// TIA Portal V17 export
// export: Created 2024-09-02T12:50:23.3039212Z, ExportSetting WithDefaults, DisplayName Totally Integrated Automation Portal, DisplayVersion V17, DisplayName TIA Portal Openness, DisplayVersion V17, DisplayName TIA Portal Version Control Interface, DisplayVersion V17, DisplayName STEP 7 Professional, DisplayVersion V17, DisplayName STEP 7 Safety, DisplayVersion V17, DisplayName WinCC Professional, DisplayVersion V17
FUNCTION "AnwFC_Aveva_OP701" : Void   // FC35, LAD
{ S7_Optimized_Access := 'TRUE' }
VERSION : 0.1
// stored: AutoNumber true, IsIECCheckEnabled false, SetENOAutomatically false, UDAEnableTagReadback false
   VAR_TEMP
      Data_Ready : Bool;
      Pallet_Nr_Moved : Bool;
      Converted_Data : Real;
      tEKSLevelOK : Bool;
   END_VAR
   VAR CONSTANT
      cButtonNotActive : USInt := 0;
      cButtonActive : USInt := 1;
      cColorRed : USInt := 2;
      cColorGreen : USInt := 3;
      cMesOptionEmpty : USInt := 0;
      cMesReasonEmpty : String := '';
   END_VAR
   VAR_TEMP   // added for the SCL form of the ladder/FBD networks
      _w1 : Bool;
      _w2 : Bool;
      _w3 : Bool;
      _w4 : Bool;
   END_VAR
BEGIN

REGION Network 1: ################STEP 1 - Pallet arrive to station #################
END_REGION

REGION Network 2: Copy Nr of Pallet
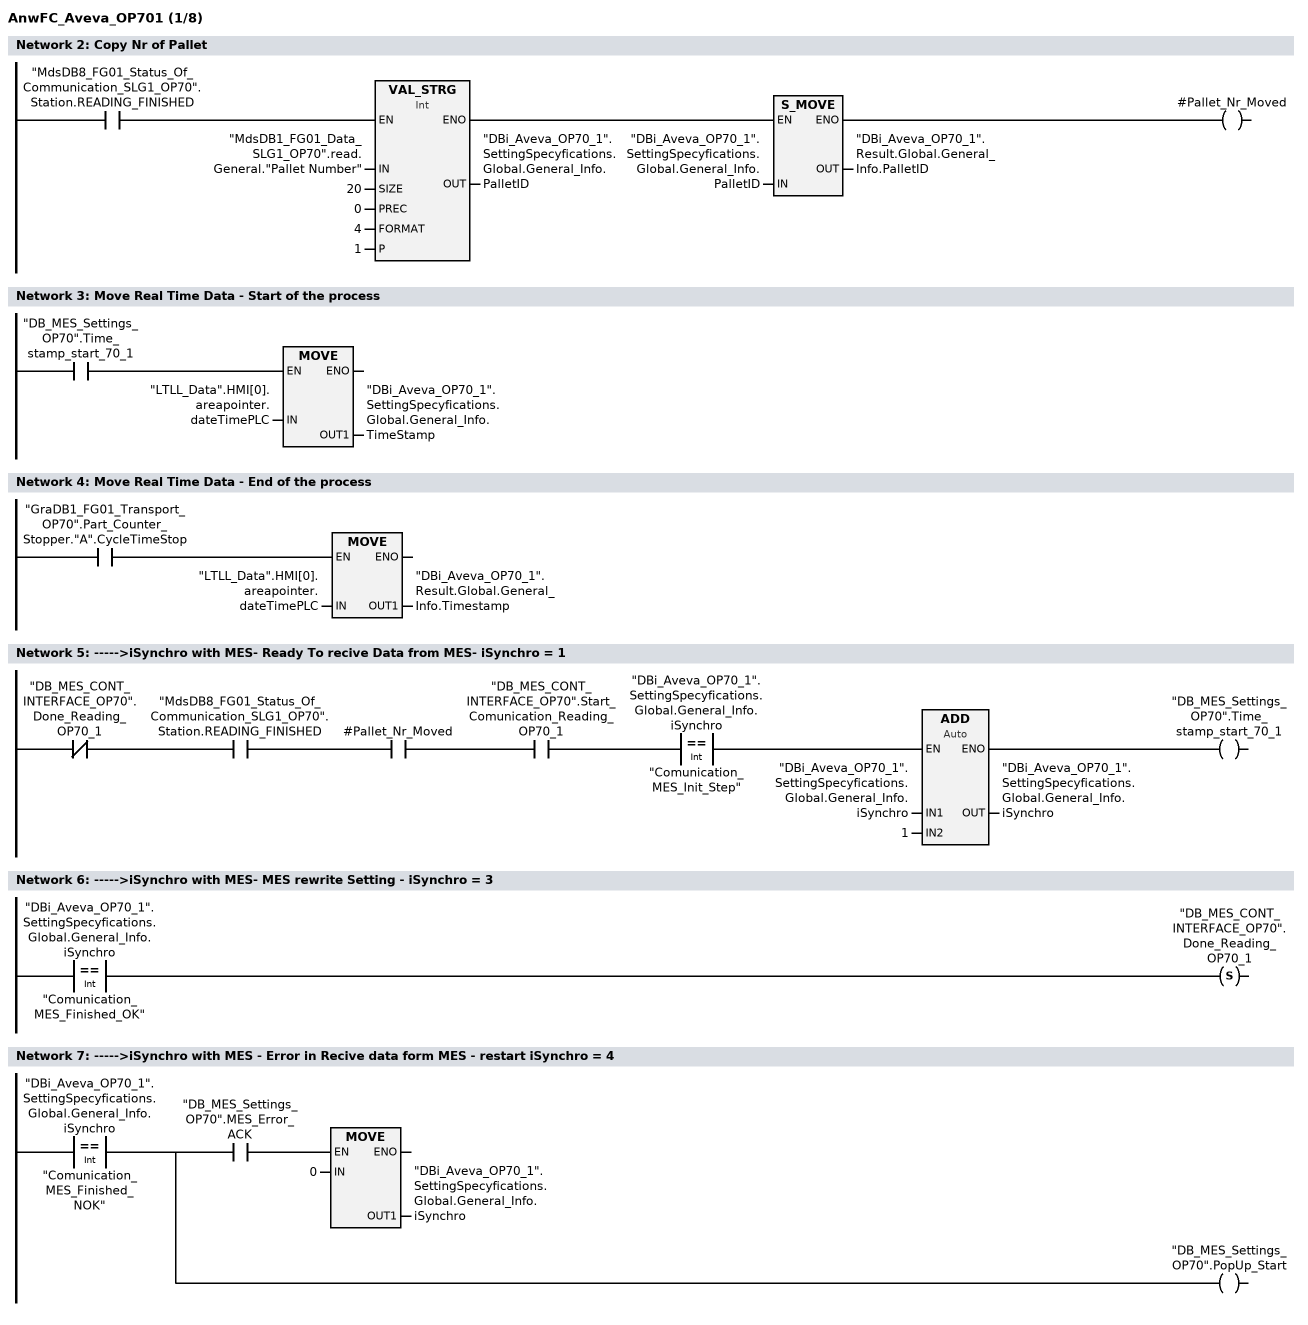
   RUNG wire#powerrail
      Contact( "MdsDB8_FG01_Status_Of_Communication_SLG1_OP70".Station.READING_FINISHED )
      { S7_Templates := "[value_type := Int, str_type := String]" } VAL_STRG(IN := "MdsDB1_FG01_Data_SLG1_OP70".read.General."Pallet Number", SIZE := 20, PREC := 0, FORMAT := 4, P := 1, OUT => "DBi_Aveva_OP70_1".SettingSpecyfications.Global.General_Info.PalletID)
      S_Move(in := "DBi_Aveva_OP70_1".SettingSpecyfications.Global.General_Info.PalletID, out => "DBi_Aveva_OP70_1".Result.Global.General_Info.PalletID)
      Coil( #Pallet_Nr_Moved )
   END_RUNG
   // the same network as SCL:
   VAL_STRG(EN := "MdsDB8_FG01_Status_Of_Communication_SLG1_OP70".Station.READING_FINISHED,
            IN := "MdsDB1_FG01_Data_SLG1_OP70".read.General."Pallet Number",
            SIZE := 20,
            PREC := 0,
            FORMAT := 4,
            P := 1,
            OUT => "DBi_Aveva_OP70_1".SettingSpecyfications.Global.General_Info.PalletID,
            ENO => #_w1);
   IF #_w1 THEN
       "DBi_Aveva_OP70_1".Result.Global.General_Info.PalletID := "DBi_Aveva_OP70_1".SettingSpecyfications.Global.General_Info.PalletID;
   END_IF;
   #Pallet_Nr_Moved := #_w1;
END_REGION

REGION Network 3: Move Real Time Data - Start of the process
   RUNG wire#powerrail
      Contact( "DB_MES_Settings_OP70".Time_stamp_start_70_1 )
      Move(in := "LTLL_Data".HMI[0].areapointer.dateTimePLC, out1 => "DBi_Aveva_OP70_1".SettingSpecyfications.Global.General_Info.TimeStamp)
   END_RUNG
   // the same network as SCL:
   IF "DB_MES_Settings_OP70".Time_stamp_start_70_1 THEN
       "DBi_Aveva_OP70_1".SettingSpecyfications.Global.General_Info.TimeStamp := "LTLL_Data".HMI[0].areapointer.dateTimePLC;
   END_IF;
END_REGION

REGION Network 4: Move Real Time Data - End of the process
   RUNG wire#powerrail
      Contact( "GraDB1_FG01_Transport_OP70".Part_Counter_Stopper."A".CycleTimeStop )
      Move(in := "LTLL_Data".HMI[0].areapointer.dateTimePLC, out1 => "DBi_Aveva_OP70_1".Result.Global.General_Info.Timestamp)
   END_RUNG
   // the same network as SCL:
   IF "GraDB1_FG01_Transport_OP70".Part_Counter_Stopper."A".CycleTimeStop THEN
       "DBi_Aveva_OP70_1".Result.Global.General_Info.Timestamp := "LTLL_Data".HMI[0].areapointer.dateTimePLC;
   END_IF;
END_REGION

REGION Network 5: ----->iSynchro with MES- Ready To recive Data from MES- iSynchro = 1
   RUNG wire#powerrail
      I_Contact( "DB_MES_CONT_INTERFACE_OP70".Done_Reading_OP70_1 )
      Contact( "MdsDB8_FG01_Status_Of_Communication_SLG1_OP70".Station.READING_FINISHED )
      Contact( #Pallet_Nr_Moved )
      Contact( "DB_MES_CONT_INTERFACE_OP70".Start_Comunication_Reading_OP70_1 )
      { S7_Templates := "SrcType := Int" } EQ_Contact(in1 := "DBi_Aveva_OP70_1".SettingSpecyfications.Global.General_Info.iSynchro, in2 := "Comunication_MES_Init_Step")
      Add(in1 := "DBi_Aveva_OP70_1".SettingSpecyfications.Global.General_Info.iSynchro, in2 := 1, out => "DBi_Aveva_OP70_1".SettingSpecyfications.Global.General_Info.iSynchro)
      Coil( "DB_MES_Settings_OP70".Time_stamp_start_70_1 )
   END_RUNG
   // the same network as SCL:
   #_w1 := NOT "DB_MES_CONT_INTERFACE_OP70".Done_Reading_OP70_1 AND "MdsDB8_FG01_Status_Of_Communication_SLG1_OP70".Station.READING_FINISHED AND #Pallet_Nr_Moved AND "DB_MES_CONT_INTERFACE_OP70".Start_Comunication_Reading_OP70_1 AND ("DBi_Aveva_OP70_1".SettingSpecyfications.Global.General_Info.iSynchro = "Comunication_MES_Init_Step");
   IF #_w1 THEN
       "DBi_Aveva_OP70_1".SettingSpecyfications.Global.General_Info.iSynchro := "DBi_Aveva_OP70_1".SettingSpecyfications.Global.General_Info.iSynchro + 1;
   END_IF;
   "DB_MES_Settings_OP70".Time_stamp_start_70_1 := #_w1;
END_REGION

REGION Network 6: ----->iSynchro with MES- MES rewrite Setting - iSynchro = 3
   RUNG wire#powerrail
      { S7_Templates := "SrcType := Int" } EQ_Contact(in1 := "DBi_Aveva_OP70_1".SettingSpecyfications.Global.General_Info.iSynchro, in2 := "Comunication_MES_Finished_OK")
      S_Coil( "DB_MES_CONT_INTERFACE_OP70".Done_Reading_OP70_1 )
   END_RUNG
   // the same network as SCL:
   IF "DBi_Aveva_OP70_1".SettingSpecyfications.Global.General_Info.iSynchro = "Comunication_MES_Finished_OK" THEN
       "DB_MES_CONT_INTERFACE_OP70".Done_Reading_OP70_1 := TRUE;
   END_IF;
END_REGION

REGION Network 7: ----->iSynchro with MES - Error in Recive data form MES - restart iSynchro = 4
   RUNG wire#powerrail
      { S7_Templates := "SrcType := Int" } EQ_Contact(in1 := "DBi_Aveva_OP70_1".SettingSpecyfications.Global.General_Info.iSynchro, in2 := "Comunication_MES_Finished_NOK")
      wire#w1
      Contact( "DB_MES_Settings_OP70".MES_Error_ACK )
      Move(in := 0, out1 => "DBi_Aveva_OP70_1".SettingSpecyfications.Global.General_Info.iSynchro)
   END_RUNG
   RUNG wire#w1
      Coil( "DB_MES_Settings_OP70".PopUp_Start )
   END_RUNG
   // the same network as SCL:
   #_w1 := "DBi_Aveva_OP70_1".SettingSpecyfications.Global.General_Info.iSynchro = "Comunication_MES_Finished_NOK";
   IF #_w1 AND "DB_MES_Settings_OP70".MES_Error_ACK THEN
       "DBi_Aveva_OP70_1".SettingSpecyfications.Global.General_Info.iSynchro := 0;
   END_IF;
   "DB_MES_Settings_OP70".PopUp_Start := #_w1;
END_REGION

REGION Network 8: ----->iSynchro with MES - End of Analyse - restart iSynchro = 0
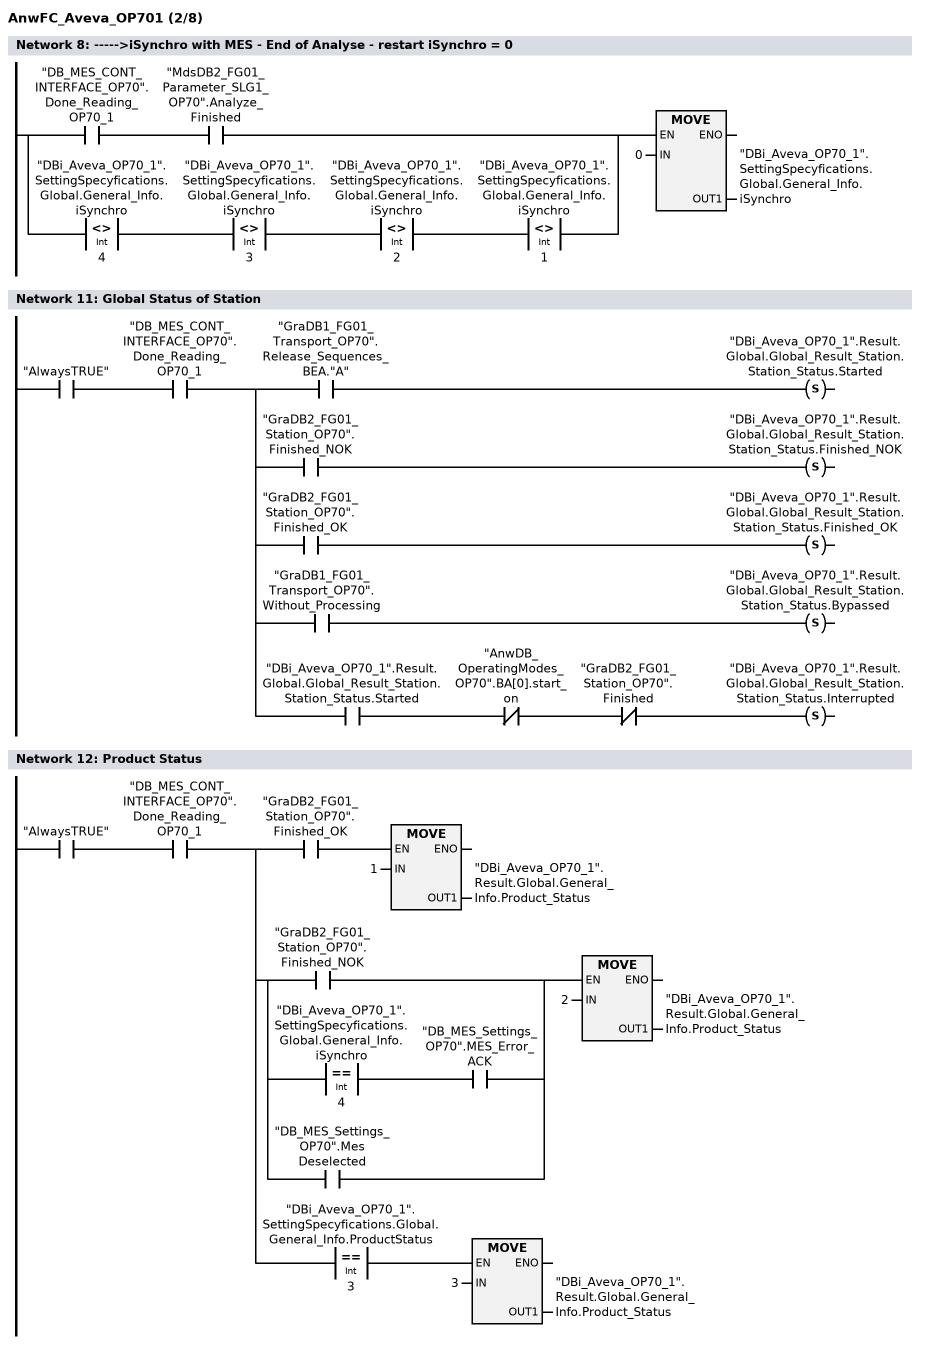
   RUNG wire#powerrail
      Contact( "DB_MES_CONT_INTERFACE_OP70".Done_Reading_OP70_1 )
      Contact( "MdsDB2_FG01_Parameter_SLG1_OP70".Analyze_Finished )
      wire#w1
      Move(in := 0, out1 => "DBi_Aveva_OP70_1".SettingSpecyfications.Global.General_Info.iSynchro)
   END_RUNG
   RUNG wire#powerrail
      { S7_Templates := "SrcType := Int" } NE_Contact(in1 := "DBi_Aveva_OP70_1".SettingSpecyfications.Global.General_Info.iSynchro, in2 := 4)
      { S7_Templates := "SrcType := Int" } NE_Contact(in1 := "DBi_Aveva_OP70_1".SettingSpecyfications.Global.General_Info.iSynchro, in2 := 3)
      { S7_Templates := "SrcType := Int" } NE_Contact(in1 := "DBi_Aveva_OP70_1".SettingSpecyfications.Global.General_Info.iSynchro, in2 := 2)
      { S7_Templates := "SrcType := Int" } NE_Contact(in1 := "DBi_Aveva_OP70_1".SettingSpecyfications.Global.General_Info.iSynchro, in2 := 1)
   END_RUNG wire#w1
   // the same network as SCL:
   IF ("DB_MES_CONT_INTERFACE_OP70".Done_Reading_OP70_1 AND "MdsDB2_FG01_Parameter_SLG1_OP70".Analyze_Finished) OR (("DBi_Aveva_OP70_1".SettingSpecyfications.Global.General_Info.iSynchro <> 4) AND ("DBi_Aveva_OP70_1".SettingSpecyfications.Global.General_Info.iSynchro <> 3) AND ("DBi_Aveva_OP70_1".SettingSpecyfications.Global.General_Info.iSynchro <> 2) AND ("DBi_Aveva_OP70_1".SettingSpecyfications.Global.General_Info.iSynchro <> 1)) THEN
       "DBi_Aveva_OP70_1".SettingSpecyfications.Global.General_Info.iSynchro := 0;
   END_IF;
END_REGION

REGION Network 9: ################STEP 2 - Move the Proce Data From Each Operation ################# / Status Proces 1
   // IN0 - Aktor ist abgewählt
   // IN1 - TAF ist angewählt
   // IN2 - Nacharbeit in Station
   // IN3 - Auftrag manuell vorgegeben
   // IN4 - Nacharbeit auf Standby-Platz
   // IN5 - Nacharbeit auf EAS-Platz
   // IN6 - TAF hat gearbeitet (Fertigmeldung)
   // IN7 - Bauteil wurde iO bearbeitet
END_REGION

REGION Network 10: ################STEP 2 - Move the Proce Data From Station ################# / Status Proces 1
   // IN0 - Aktor ist abgewählt
   // IN1 - TAF ist angewählt
   // IN2 - Nacharbeit in Station
   // IN3 - Auftrag manuell vorgegeben
   // IN4 - Nacharbeit auf Standby-Platz
   // IN5 - Nacharbeit auf EAS-Platz
   // IN6 - TAF hat gearbeitet (Fertigmeldung)
   // IN7 - Bauteil wurde iO bearbeitet
END_REGION

REGION Network 11: Global Status of Station
   RUNG wire#powerrail
      Contact( "AlwaysTRUE" )
      Contact( "DB_MES_CONT_INTERFACE_OP70".Done_Reading_OP70_1 )
      wire#w1
      Contact( "GraDB1_FG01_Transport_OP70".Release_Sequences_BEA."A" )
      S_Coil( "DBi_Aveva_OP70_1".Result.Global.Global_Result_Station.Station_Status.Started )
   END_RUNG
   RUNG wire#w1
      Contact( "GraDB2_FG01_Station_OP70".Finished_NOK )
      S_Coil( "DBi_Aveva_OP70_1".Result.Global.Global_Result_Station.Station_Status.Finished_NOK )
   END_RUNG
   RUNG wire#w1
      Contact( "GraDB2_FG01_Station_OP70".Finished_OK )
      S_Coil( "DBi_Aveva_OP70_1".Result.Global.Global_Result_Station.Station_Status.Finished_OK )
   END_RUNG
   RUNG wire#w1
      Contact( "GraDB1_FG01_Transport_OP70".Without_Processing )
      S_Coil( "DBi_Aveva_OP70_1".Result.Global.Global_Result_Station.Station_Status.Bypassed )
   END_RUNG
   RUNG wire#w1
      Contact( "DBi_Aveva_OP70_1".Result.Global.Global_Result_Station.Station_Status.Started )
      I_Contact( "AnwDB_OperatingModes_OP70".BA[0].start_on )
      I_Contact( "GraDB2_FG01_Station_OP70".Finished )
      S_Coil( "DBi_Aveva_OP70_1".Result.Global.Global_Result_Station.Station_Status.Interrupted )
   END_RUNG
   // the same network as SCL:
   #_w1 := "AlwaysTRUE" AND "DB_MES_CONT_INTERFACE_OP70".Done_Reading_OP70_1;
   IF #_w1 AND "GraDB1_FG01_Transport_OP70".Release_Sequences_BEA."A" THEN
       "DBi_Aveva_OP70_1".Result.Global.Global_Result_Station.Station_Status.Started := TRUE;
   END_IF;
   IF #_w1 AND "GraDB2_FG01_Station_OP70".Finished_NOK THEN
       "DBi_Aveva_OP70_1".Result.Global.Global_Result_Station.Station_Status.Finished_NOK := TRUE;
   END_IF;
   IF #_w1 AND "GraDB2_FG01_Station_OP70".Finished_OK THEN
       "DBi_Aveva_OP70_1".Result.Global.Global_Result_Station.Station_Status.Finished_OK := TRUE;
   END_IF;
   IF #_w1 AND "GraDB1_FG01_Transport_OP70".Without_Processing THEN
       "DBi_Aveva_OP70_1".Result.Global.Global_Result_Station.Station_Status.Bypassed := TRUE;
   END_IF;
   IF #_w1 AND "DBi_Aveva_OP70_1".Result.Global.Global_Result_Station.Station_Status.Started AND NOT "AnwDB_OperatingModes_OP70".BA[0].start_on AND NOT "GraDB2_FG01_Station_OP70".Finished THEN
       "DBi_Aveva_OP70_1".Result.Global.Global_Result_Station.Station_Status.Interrupted := TRUE;
   END_IF;
END_REGION

REGION Network 12: Product Status
   RUNG wire#powerrail
      Contact( "AlwaysTRUE" )
      Contact( "DB_MES_CONT_INTERFACE_OP70".Done_Reading_OP70_1 )
      wire#w1
      Contact( "GraDB2_FG01_Station_OP70".Finished_OK )
      Move(in := 1, out1 => "DBi_Aveva_OP70_1".Result.Global.General_Info.Product_Status)
   END_RUNG
   RUNG wire#w1
      Contact( "GraDB2_FG01_Station_OP70".Finished_NOK )
      wire#w2
      Move(in := 2, out1 => "DBi_Aveva_OP70_1".Result.Global.General_Info.Product_Status)
   END_RUNG
   RUNG wire#w1
      { S7_Templates := "SrcType := Int" } EQ_Contact(in1 := "DBi_Aveva_OP70_1".SettingSpecyfications.Global.General_Info.iSynchro, in2 := 4)
      Contact( "DB_MES_Settings_OP70".MES_Error_ACK )
   END_RUNG wire#w2
   RUNG wire#w1
      Contact( "DB_MES_Settings_OP70".MesDeselected )
   END_RUNG wire#w2
   RUNG wire#w1
      { S7_Templates := "SrcType := Int" } EQ_Contact(in1 := "DBi_Aveva_OP70_1".SettingSpecyfications.Global.General_Info.ProductStatus, in2 := 3)
      Move(in := 3, out1 => "DBi_Aveva_OP70_1".Result.Global.General_Info.Product_Status)
   END_RUNG
   // the same network as SCL:
   #_w1 := "AlwaysTRUE" AND "DB_MES_CONT_INTERFACE_OP70".Done_Reading_OP70_1;
   IF #_w1 AND "GraDB2_FG01_Station_OP70".Finished_OK THEN
       "DBi_Aveva_OP70_1".Result.Global.General_Info.Product_Status := 1;
   END_IF;
   IF #_w1 AND ("GraDB2_FG01_Station_OP70".Finished_NOK OR (("DBi_Aveva_OP70_1".SettingSpecyfications.Global.General_Info.iSynchro = 4) AND "DB_MES_Settings_OP70".MES_Error_ACK) OR "DB_MES_Settings_OP70".MesDeselected) THEN
       "DBi_Aveva_OP70_1".Result.Global.General_Info.Product_Status := 2;
   END_IF;
   IF #_w1 AND ("DBi_Aveva_OP70_1".SettingSpecyfications.Global.General_Info.ProductStatus = 3) THEN
       "DBi_Aveva_OP70_1".Result.Global.General_Info.Product_Status := 3;
   END_IF;
END_REGION

REGION Network 13: ################ STEP 3 - Prepare Isynchro for MES in result area #################
END_REGION

REGION Network 14: ----->iSynchro with MES- Ready To copy Data to MES- - iSynchro = 1
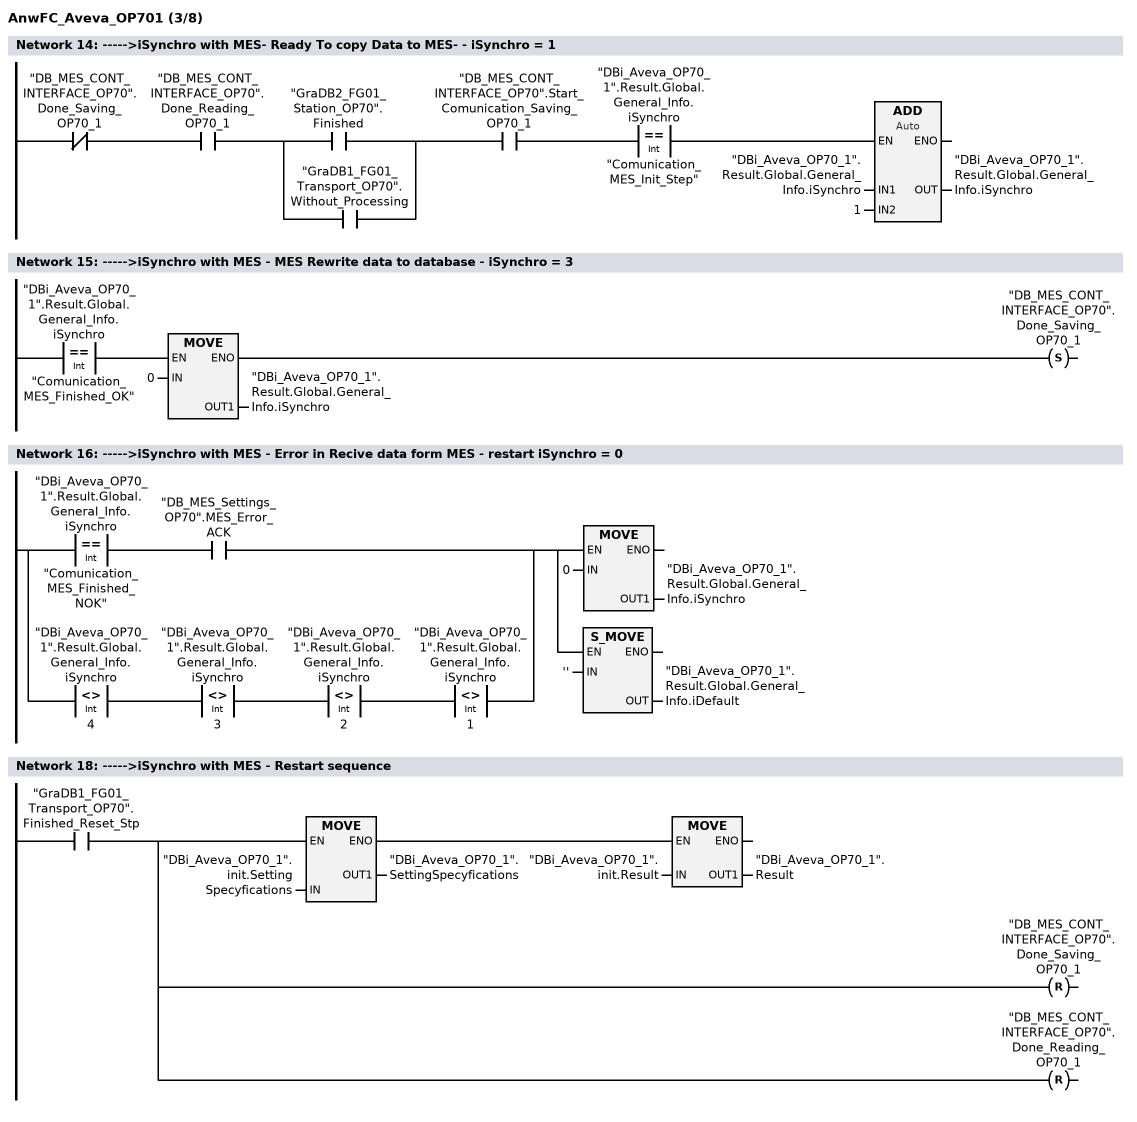
   RUNG wire#powerrail
      I_Contact( "DB_MES_CONT_INTERFACE_OP70".Done_Saving_OP70_1 )
      Contact( "DB_MES_CONT_INTERFACE_OP70".Done_Reading_OP70_1 )
      wire#w1
      Contact( "GraDB2_FG01_Station_OP70".Finished )
      wire#w2
      Contact( "DB_MES_CONT_INTERFACE_OP70".Start_Comunication_Saving_OP70_1 )
      { S7_Templates := "SrcType := Int" } EQ_Contact(in1 := "DBi_Aveva_OP70_1".Result.Global.General_Info.iSynchro, in2 := "Comunication_MES_Init_Step")
      Add(in1 := "DBi_Aveva_OP70_1".Result.Global.General_Info.iSynchro, in2 := 1, out => "DBi_Aveva_OP70_1".Result.Global.General_Info.iSynchro)
   END_RUNG
   RUNG wire#w1
      Contact( "GraDB1_FG01_Transport_OP70".Without_Processing )
   END_RUNG wire#w2
   // the same network as SCL:
   IF NOT "DB_MES_CONT_INTERFACE_OP70".Done_Saving_OP70_1 AND "DB_MES_CONT_INTERFACE_OP70".Done_Reading_OP70_1 AND ("GraDB2_FG01_Station_OP70".Finished OR "GraDB1_FG01_Transport_OP70".Without_Processing) AND "DB_MES_CONT_INTERFACE_OP70".Start_Comunication_Saving_OP70_1 AND ("DBi_Aveva_OP70_1".Result.Global.General_Info.iSynchro = "Comunication_MES_Init_Step") THEN
       "DBi_Aveva_OP70_1".Result.Global.General_Info.iSynchro := "DBi_Aveva_OP70_1".Result.Global.General_Info.iSynchro + 1;
   END_IF;
END_REGION

REGION Network 15: ----->iSynchro with MES - MES Rewrite data to database - iSynchro = 3
   RUNG wire#powerrail
      { S7_Templates := "SrcType := Int" } EQ_Contact(in1 := "DBi_Aveva_OP70_1".Result.Global.General_Info.iSynchro, in2 := "Comunication_MES_Finished_OK")
      Move(in := 0, out1 => "DBi_Aveva_OP70_1".Result.Global.General_Info.iSynchro)
      S_Coil( "DB_MES_CONT_INTERFACE_OP70".Done_Saving_OP70_1 )
   END_RUNG
   // the same network as SCL:
   #_w1 := "DBi_Aveva_OP70_1".Result.Global.General_Info.iSynchro = "Comunication_MES_Finished_OK";
   IF #_w1 THEN
       "DBi_Aveva_OP70_1".Result.Global.General_Info.iSynchro := 0;
       "DB_MES_CONT_INTERFACE_OP70".Done_Saving_OP70_1 := TRUE;
   END_IF;
END_REGION

REGION Network 16: ----->iSynchro with MES - Error in Recive data form MES - restart iSynchro = 0
   RUNG wire#powerrail
      { S7_Templates := "SrcType := Int" } EQ_Contact(in1 := "DBi_Aveva_OP70_1".Result.Global.General_Info.iSynchro, in2 := "Comunication_MES_Finished_NOK")
      Contact( "DB_MES_Settings_OP70".MES_Error_ACK )
      wire#w1
      Move(in := 0, out1 => "DBi_Aveva_OP70_1".Result.Global.General_Info.iSynchro)
   END_RUNG
   RUNG wire#powerrail
      { S7_Templates := "SrcType := Int" } NE_Contact(in1 := "DBi_Aveva_OP70_1".Result.Global.General_Info.iSynchro, in2 := 4)
      { S7_Templates := "SrcType := Int" } NE_Contact(in1 := "DBi_Aveva_OP70_1".Result.Global.General_Info.iSynchro, in2 := 3)
      { S7_Templates := "SrcType := Int" } NE_Contact(in1 := "DBi_Aveva_OP70_1".Result.Global.General_Info.iSynchro, in2 := 2)
      { S7_Templates := "SrcType := Int" } NE_Contact(in1 := "DBi_Aveva_OP70_1".Result.Global.General_Info.iSynchro, in2 := 1)
   END_RUNG wire#w1
   RUNG wire#w1
      S_Move(in := '', out => "DBi_Aveva_OP70_1".Result.Global.General_Info.iDefault)
   END_RUNG
   // the same network as SCL:
   #_w1 := (("DBi_Aveva_OP70_1".Result.Global.General_Info.iSynchro = "Comunication_MES_Finished_NOK") AND "DB_MES_Settings_OP70".MES_Error_ACK) OR (("DBi_Aveva_OP70_1".Result.Global.General_Info.iSynchro <> 4) AND ("DBi_Aveva_OP70_1".Result.Global.General_Info.iSynchro <> 3) AND ("DBi_Aveva_OP70_1".Result.Global.General_Info.iSynchro <> 2) AND ("DBi_Aveva_OP70_1".Result.Global.General_Info.iSynchro <> 1));
   IF #_w1 THEN
       "DBi_Aveva_OP70_1".Result.Global.General_Info.iSynchro := 0;
       "DBi_Aveva_OP70_1".Result.Global.General_Info.iDefault := '';
   END_IF;
END_REGION

REGION Network 17: ################ STEP3 - Restart all #################
END_REGION

REGION Network 18: ----->iSynchro with MES - Restart sequence
   RUNG wire#powerrail
      Contact( "GraDB1_FG01_Transport_OP70".Finished_Reset_Stp )
      wire#w1
      Move(in := "DBi_Aveva_OP70_1".init.SettingSpecyfications, out1 => "DBi_Aveva_OP70_1".SettingSpecyfications)
      Move(in := "DBi_Aveva_OP70_1".init.Result, out1 => "DBi_Aveva_OP70_1".Result)
   END_RUNG
   RUNG wire#w1
      R_Coil( "DB_MES_CONT_INTERFACE_OP70".Done_Saving_OP70_1 )
   END_RUNG
   RUNG wire#w1
      R_Coil( "DB_MES_CONT_INTERFACE_OP70".Done_Reading_OP70_1 )
   END_RUNG
   // the same network as SCL:
   IF "GraDB1_FG01_Transport_OP70".Finished_Reset_Stp THEN
       "DBi_Aveva_OP70_1".SettingSpecyfications := "DBi_Aveva_OP70_1".init.SettingSpecyfications;
       "DBi_Aveva_OP70_1".Result := "DBi_Aveva_OP70_1".init.Result;
       "DB_MES_CONT_INTERFACE_OP70".Done_Saving_OP70_1 := FALSE;
       "DB_MES_CONT_INTERFACE_OP70".Done_Reading_OP70_1 := FALSE;
   END_IF;
END_REGION

REGION Network 19: ################ Status of machine #################
END_REGION

REGION Network 20: Auto/ Hand/ Station started/ Error
   // %X0 - (WS)Media ON, 
   // %X1 - (WS)Hand selected,
   // %X2 - (WS)Auto selected, 
   // %X3 - (WS)Start ON(with auto or hand Mode),  
   // %X4 - (WS)Error,  
   // %X5 - (WS)Clock_1Hz - lifebit, 
   // %X6 - (MES)Clock_1Hz - lifebit ,  
   // %X7 - (MES)Automatic on Conveyor
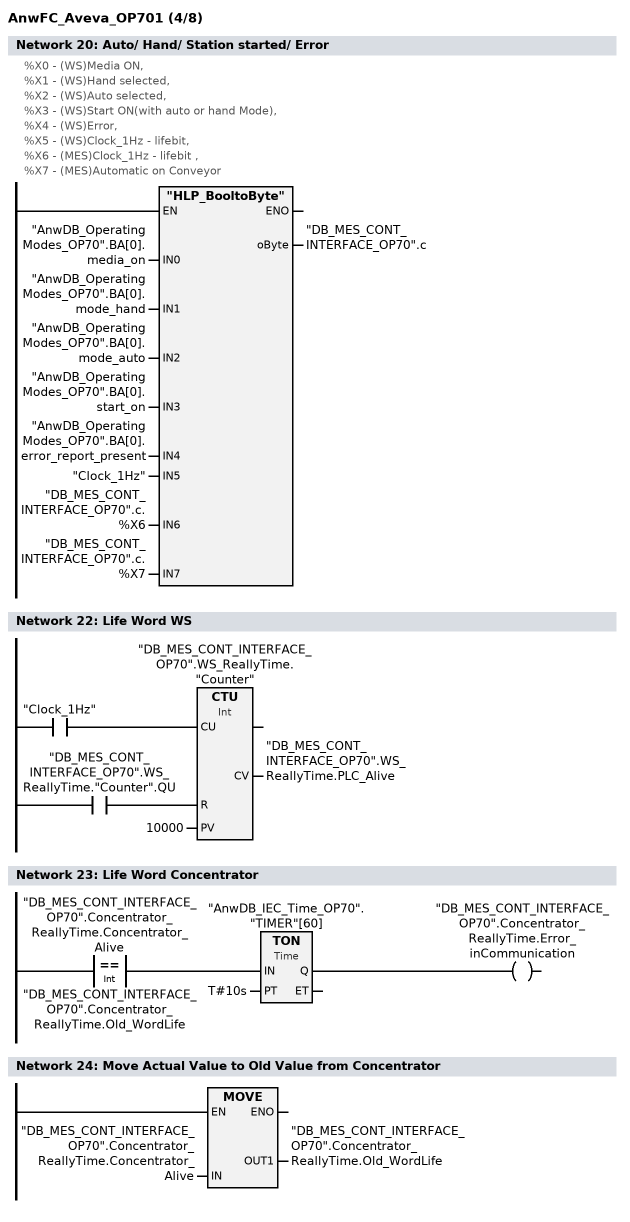
   RUNG wire#powerrail
      "HLP_BooltoByte"(IN0 := "AnwDB_OperatingModes_OP70".BA[0].media_on, IN1 := "AnwDB_OperatingModes_OP70".BA[0].mode_hand, IN2 := "AnwDB_OperatingModes_OP70".BA[0].mode_auto, IN3 := "AnwDB_OperatingModes_OP70".BA[0].start_on, IN4 := "AnwDB_OperatingModes_OP70".BA[0].error_report_present, IN5 := "Clock_1Hz", IN6 := "DB_MES_CONT_INTERFACE_OP70".c.%X6, IN7 := "DB_MES_CONT_INTERFACE_OP70".c.%X7, oByte => "DB_MES_CONT_INTERFACE_OP70".c)
   END_RUNG
   // the same network as SCL:
   "HLP_BooltoByte"(IN0 := "AnwDB_OperatingModes_OP70".BA[0].media_on,
                    IN1 := "AnwDB_OperatingModes_OP70".BA[0].mode_hand,
                    IN2 := "AnwDB_OperatingModes_OP70".BA[0].mode_auto,
                    IN3 := "AnwDB_OperatingModes_OP70".BA[0].start_on,
                    IN4 := "AnwDB_OperatingModes_OP70".BA[0].error_report_present,
                    IN5 := "Clock_1Hz",
                    IN6 := "DB_MES_CONT_INTERFACE_OP70".c.%X6,
                    IN7 := "DB_MES_CONT_INTERFACE_OP70".c.%X7,
                    oByte => "DB_MES_CONT_INTERFACE_OP70".c);
END_REGION

REGION Network 21: ################ Communication Status #################
END_REGION

REGION Network 22: Life Word WS
   RUNG wire#powerrail
      Contact( "Clock_1Hz" )
      { S7_Templates := "value_type := Int" } "DB_MES_CONT_INTERFACE_OP70".WS_ReallyTime."Counter".CTU(r := wire#w1, pv := 10000, cv => "DB_MES_CONT_INTERFACE_OP70".WS_ReallyTime.PLC_Alive)
   END_RUNG
   RUNG wire#powerrail
      Contact( "DB_MES_CONT_INTERFACE_OP70".WS_ReallyTime."Counter".QU )
   END_RUNG wire#w1
   // the same network as SCL:
   "DB_MES_CONT_INTERFACE_OP70".WS_ReallyTime."Counter".CTU(CU := "Clock_1Hz",
                           R := "DB_MES_CONT_INTERFACE_OP70".WS_ReallyTime."Counter".QU,
                           PV := 10000,
                           CV => "DB_MES_CONT_INTERFACE_OP70".WS_ReallyTime.PLC_Alive);
END_REGION

REGION Network 23: Life Word Concentrator
   RUNG wire#powerrail
      { S7_Templates := "SrcType := Int" } EQ_Contact(in1 := "DB_MES_CONT_INTERFACE_OP70".Concentrator_ReallyTime.Concentrator_Alive, in2 := "DB_MES_CONT_INTERFACE_OP70".Concentrator_ReallyTime.Old_WordLife)
      { S7_Templates := "time_type := Time" } "AnwDB_IEC_Time_OP70"."TIMER"[60].TON(pt := T#10s, et =>)
      Coil( "DB_MES_CONT_INTERFACE_OP70".Concentrator_ReallyTime.Error_inCommunication )
   END_RUNG
   // the same network as SCL:
   "AnwDB_IEC_Time_OP70"."TIMER"[60].TON(IN := "DB_MES_CONT_INTERFACE_OP70".Concentrator_ReallyTime.Concentrator_Alive = "DB_MES_CONT_INTERFACE_OP70".Concentrator_ReallyTime.Old_WordLife,
                           PT := T#10s);
   "DB_MES_CONT_INTERFACE_OP70".Concentrator_ReallyTime.Error_inCommunication := "AnwDB_IEC_Time_OP70"."TIMER"[60].Q;
END_REGION

REGION Network 24: Move Actual Value to Old Value from Concentrator
   RUNG wire#powerrail
      Move(in := "DB_MES_CONT_INTERFACE_OP70".Concentrator_ReallyTime.Concentrator_Alive, out1 => "DB_MES_CONT_INTERFACE_OP70".Concentrator_ReallyTime.Old_WordLife)
   END_RUNG
   // the same network as SCL:
   "DB_MES_CONT_INTERFACE_OP70".Concentrator_ReallyTime.Old_WordLife := "DB_MES_CONT_INTERFACE_OP70".Concentrator_ReallyTime.Concentrator_Alive;
END_REGION

REGION Network 25: isynchro test - Delate
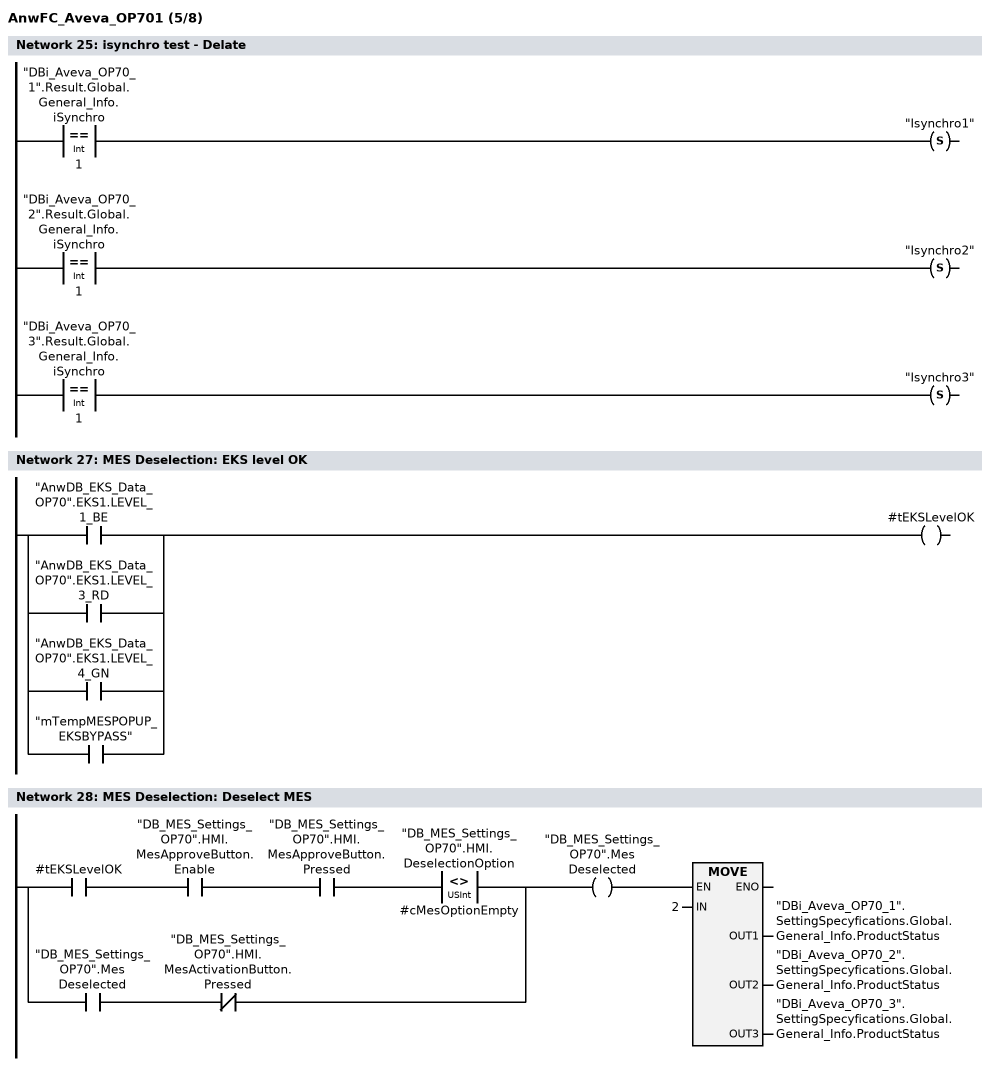
   RUNG wire#powerrail
      { S7_Templates := "SrcType := Int" } EQ_Contact(in1 := "DBi_Aveva_OP70_1".Result.Global.General_Info.iSynchro, in2 := 1)
      S_Coil( "Isynchro1" )
   END_RUNG
   RUNG wire#powerrail
      { S7_Templates := "SrcType := Int" } EQ_Contact(in1 := "DBi_Aveva_OP70_2".Result.Global.General_Info.iSynchro, in2 := 1)
      S_Coil( "Isynchro2" )
   END_RUNG
   RUNG wire#powerrail
      { S7_Templates := "SrcType := Int" } EQ_Contact(in1 := "DBi_Aveva_OP70_3".Result.Global.General_Info.iSynchro, in2 := 1)
      S_Coil( "Isynchro3" )
   END_RUNG
   // the same network as SCL:
   IF "DBi_Aveva_OP70_1".Result.Global.General_Info.iSynchro = 1 THEN "Isynchro1" := TRUE; END_IF;
   IF "DBi_Aveva_OP70_2".Result.Global.General_Info.iSynchro = 1 THEN "Isynchro2" := TRUE; END_IF;
   IF "DBi_Aveva_OP70_3".Result.Global.General_Info.iSynchro = 1 THEN "Isynchro3" := TRUE; END_IF;
END_REGION

REGION Network 26: ################ MES DESELECTION #################
END_REGION

REGION Network 27: MES Deselection: EKS level OK
   RUNG wire#powerrail
      Contact( "AnwDB_EKS_Data_OP70".EKS1.LEVEL_1_BE )
      wire#w1
      Coil( #tEKSLevelOK )
   END_RUNG
   RUNG wire#powerrail
      Contact( "AnwDB_EKS_Data_OP70".EKS1.LEVEL_3_RD )
   END_RUNG wire#w1
   RUNG wire#powerrail
      Contact( "AnwDB_EKS_Data_OP70".EKS1.LEVEL_4_GN )
   END_RUNG wire#w1
   RUNG wire#powerrail
      Contact( "mTempMESPOPUP_EKSBYPASS" )
   END_RUNG wire#w1
   // the same network as SCL:
   #tEKSLevelOK := "AnwDB_EKS_Data_OP70".EKS1.LEVEL_1_BE OR "AnwDB_EKS_Data_OP70".EKS1.LEVEL_3_RD OR "AnwDB_EKS_Data_OP70".EKS1.LEVEL_4_GN OR "mTempMESPOPUP_EKSBYPASS";
END_REGION

REGION Network 28: MES Deselection: Deselect MES
   RUNG wire#powerrail
      Contact( #tEKSLevelOK )
      Contact( "DB_MES_Settings_OP70".HMI.MesApproveButton.Enable )
      Contact( "DB_MES_Settings_OP70".HMI.MesApproveButton.Pressed )
      { S7_Templates := "SrcType := USInt" } NE_Contact(in1 := "DB_MES_Settings_OP70".HMI.DeselectionOption, in2 := #cMesOptionEmpty)
      wire#w1
      Coil( "DB_MES_Settings_OP70".MesDeselected )
      Move(in := 2, out1 => "DBi_Aveva_OP70_1".SettingSpecyfications.Global.General_Info.ProductStatus, out2 => "DBi_Aveva_OP70_2".SettingSpecyfications.Global.General_Info.ProductStatus, out3 => "DBi_Aveva_OP70_3".SettingSpecyfications.Global.General_Info.ProductStatus)
   END_RUNG
   RUNG wire#powerrail
      Contact( "DB_MES_Settings_OP70".MesDeselected )
      I_Contact( "DB_MES_Settings_OP70".HMI.MesActivationButton.Pressed )
   END_RUNG wire#w1
   // the same network as SCL:
   "DB_MES_Settings_OP70".MesDeselected := (#tEKSLevelOK AND "DB_MES_Settings_OP70".HMI.MesApproveButton.Enable AND "DB_MES_Settings_OP70".HMI.MesApproveButton.Pressed AND ("DB_MES_Settings_OP70".HMI.DeselectionOption <> #cMesOptionEmpty)) OR ("DB_MES_Settings_OP70".MesDeselected AND NOT "DB_MES_Settings_OP70".HMI.MesActivationButton.Pressed);
   IF "DB_MES_Settings_OP70".MesDeselected THEN
       "DBi_Aveva_OP70_1".SettingSpecyfications.Global.General_Info.ProductStatus := 2;
       "DBi_Aveva_OP70_2".SettingSpecyfications.Global.General_Info.ProductStatus := 2;
       "DBi_Aveva_OP70_3".SettingSpecyfications.Global.General_Info.ProductStatus := 2;
   END_IF;
END_REGION

REGION Network 29: MES Deselection: Send deselection reason to MES
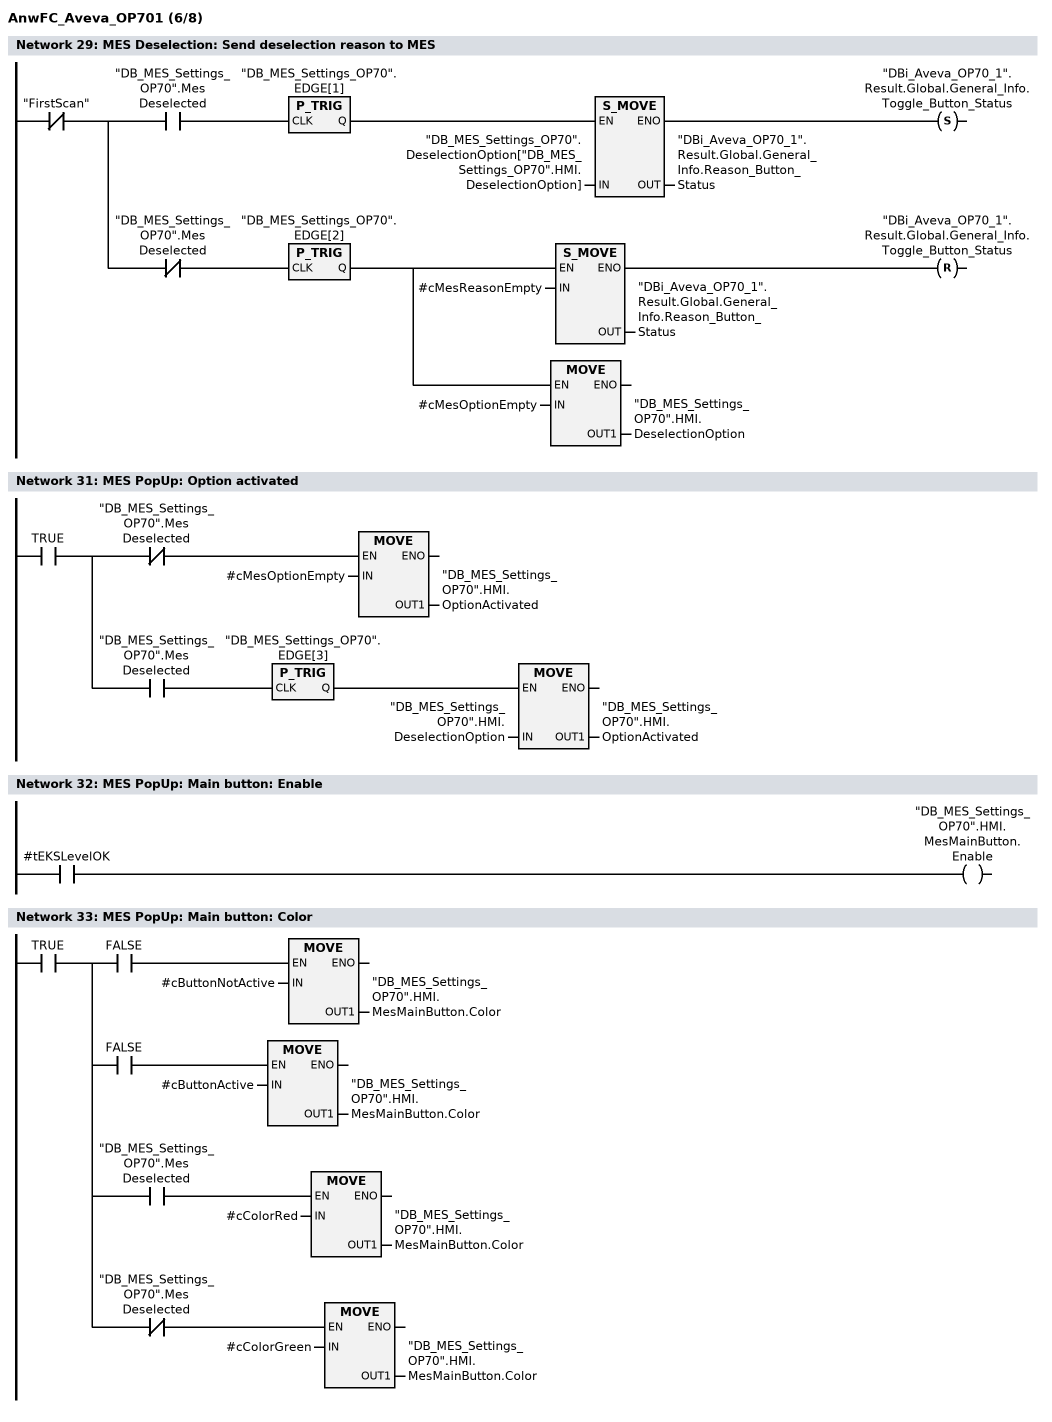
   RUNG wire#powerrail
      I_Contact( "FirstScan" )
      wire#w1
      Contact( "DB_MES_Settings_OP70".MesDeselected )
      P_Trig( "DB_MES_Settings_OP70".EDGE[1] )
      S_Move(in := "DB_MES_Settings_OP70".DeselectionOption["DB_MES_Settings_OP70".HMI.DeselectionOption], out => "DBi_Aveva_OP70_1".Result.Global.General_Info.Reason_Button_Status)
      S_Coil( "DBi_Aveva_OP70_1".Result.Global.General_Info.Toggle_Button_Status )
   END_RUNG
   RUNG wire#w1
      I_Contact( "DB_MES_Settings_OP70".MesDeselected )
      P_Trig( "DB_MES_Settings_OP70".EDGE[2] )
      wire#w2
      S_Move(in := #cMesReasonEmpty, out => "DBi_Aveva_OP70_1".Result.Global.General_Info.Reason_Button_Status)
      R_Coil( "DBi_Aveva_OP70_1".Result.Global.General_Info.Toggle_Button_Status )
   END_RUNG
   RUNG wire#w2
      Move(in := #cMesOptionEmpty, out1 => "DB_MES_Settings_OP70".HMI.DeselectionOption)
   END_RUNG
   // the same network as SCL:
   #_w1 := NOT "FirstScan" AND "DB_MES_Settings_OP70".MesDeselected;
   #_w2 := #_w1 AND NOT "DB_MES_Settings_OP70".EDGE[1];   // rising edge
   "DB_MES_Settings_OP70".EDGE[1] := #_w1;
   IF #_w2 THEN
       "DBi_Aveva_OP70_1".Result.Global.General_Info.Reason_Button_Status := "DB_MES_Settings_OP70".DeselectionOption["DB_MES_Settings_OP70".HMI.DeselectionOption];
       "DBi_Aveva_OP70_1".Result.Global.General_Info.Toggle_Button_Status := TRUE;
   END_IF;
   #_w3 := NOT "FirstScan" AND NOT "DB_MES_Settings_OP70".MesDeselected;
   #_w4 := #_w3 AND NOT "DB_MES_Settings_OP70".EDGE[2];   // rising edge
   "DB_MES_Settings_OP70".EDGE[2] := #_w3;
   IF #_w4 THEN
       "DBi_Aveva_OP70_1".Result.Global.General_Info.Reason_Button_Status := #cMesReasonEmpty;
       "DBi_Aveva_OP70_1".Result.Global.General_Info.Toggle_Button_Status := FALSE;
       "DB_MES_Settings_OP70".HMI.DeselectionOption := #cMesOptionEmpty;
   END_IF;
END_REGION

REGION Network 30: ################ MES POPUP #################
END_REGION

REGION Network 31: MES PopUp: Option activated
   RUNG wire#powerrail
      Contact( TRUE )
      wire#w1
      I_Contact( "DB_MES_Settings_OP70".MesDeselected )
      Move(in := #cMesOptionEmpty, out1 => "DB_MES_Settings_OP70".HMI.OptionActivated)
   END_RUNG
   RUNG wire#w1
      Contact( "DB_MES_Settings_OP70".MesDeselected )
      P_Trig( "DB_MES_Settings_OP70".EDGE[3] )
      Move(in := "DB_MES_Settings_OP70".HMI.DeselectionOption, out1 => "DB_MES_Settings_OP70".HMI.OptionActivated)
   END_RUNG
   // the same network as SCL:
   IF TRUE AND NOT "DB_MES_Settings_OP70".MesDeselected THEN
       "DB_MES_Settings_OP70".HMI.OptionActivated := #cMesOptionEmpty;
   END_IF;
   #_w1 := TRUE AND "DB_MES_Settings_OP70".MesDeselected;
   #_w2 := #_w1 AND NOT "DB_MES_Settings_OP70".EDGE[3];   // rising edge
   "DB_MES_Settings_OP70".EDGE[3] := #_w1;
   IF #_w2 THEN
       "DB_MES_Settings_OP70".HMI.OptionActivated := "DB_MES_Settings_OP70".HMI.DeselectionOption;
   END_IF;
END_REGION

REGION Network 32: MES PopUp: Main button: Enable
   RUNG wire#powerrail
      Contact( #tEKSLevelOK )
      Coil( "DB_MES_Settings_OP70".HMI.MesMainButton.Enable )
   END_RUNG
   // the same network as SCL:
   "DB_MES_Settings_OP70".HMI.MesMainButton.Enable := #tEKSLevelOK;
END_REGION

REGION Network 33: MES PopUp: Main button: Color
   RUNG wire#powerrail
      Contact( TRUE )
      wire#w1
      Contact( FALSE )
      Move(in := #cButtonNotActive, out1 => "DB_MES_Settings_OP70".HMI.MesMainButton.Color)
   END_RUNG
   RUNG wire#w1
      Contact( FALSE )
      Move(in := #cButtonActive, out1 => "DB_MES_Settings_OP70".HMI.MesMainButton.Color)
   END_RUNG
   RUNG wire#w1
      Contact( "DB_MES_Settings_OP70".MesDeselected )
      Move(in := #cColorRed, out1 => "DB_MES_Settings_OP70".HMI.MesMainButton.Color)
   END_RUNG
   RUNG wire#w1
      I_Contact( "DB_MES_Settings_OP70".MesDeselected )
      Move(in := #cColorGreen, out1 => "DB_MES_Settings_OP70".HMI.MesMainButton.Color)
   END_RUNG
   // the same network as SCL:
   IF TRUE AND FALSE THEN
       "DB_MES_Settings_OP70".HMI.MesMainButton.Color := #cButtonNotActive;
       "DB_MES_Settings_OP70".HMI.MesMainButton.Color := #cButtonActive;
   END_IF;
   IF TRUE AND "DB_MES_Settings_OP70".MesDeselected THEN
       "DB_MES_Settings_OP70".HMI.MesMainButton.Color := #cColorRed;
   END_IF;
   IF TRUE AND NOT "DB_MES_Settings_OP70".MesDeselected THEN
       "DB_MES_Settings_OP70".HMI.MesMainButton.Color := #cColorGreen;
   END_IF;
END_REGION

REGION Network 34: MES PopUp: Approve button: Enable
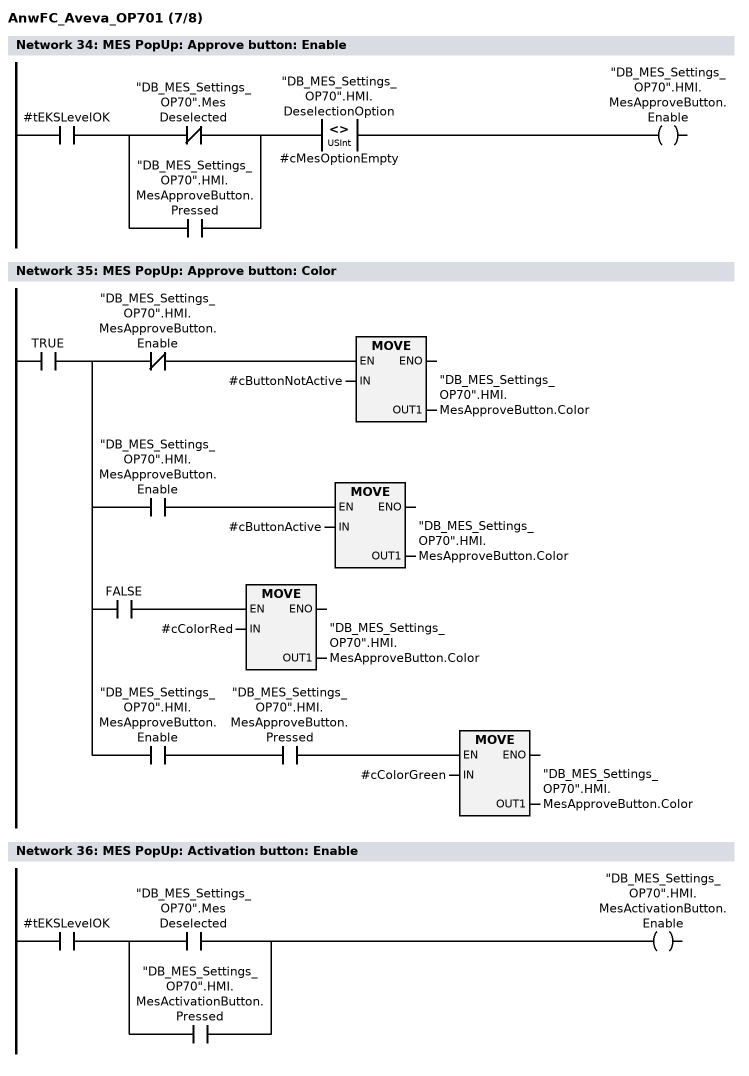
   RUNG wire#powerrail
      Contact( #tEKSLevelOK )
      wire#w1
      I_Contact( "DB_MES_Settings_OP70".MesDeselected )
      wire#w2
      { S7_Templates := "SrcType := USInt" } NE_Contact(in1 := "DB_MES_Settings_OP70".HMI.DeselectionOption, in2 := #cMesOptionEmpty)
      Coil( "DB_MES_Settings_OP70".HMI.MesApproveButton.Enable )
   END_RUNG
   RUNG wire#w1
      Contact( "DB_MES_Settings_OP70".HMI.MesApproveButton.Pressed )
   END_RUNG wire#w2
   // the same network as SCL:
   "DB_MES_Settings_OP70".HMI.MesApproveButton.Enable := #tEKSLevelOK AND (NOT "DB_MES_Settings_OP70".MesDeselected OR "DB_MES_Settings_OP70".HMI.MesApproveButton.Pressed) AND ("DB_MES_Settings_OP70".HMI.DeselectionOption <> #cMesOptionEmpty);
END_REGION

REGION Network 35: MES PopUp: Approve button: Color
   RUNG wire#powerrail
      Contact( TRUE )
      wire#w1
      I_Contact( "DB_MES_Settings_OP70".HMI.MesApproveButton.Enable )
      Move(in := #cButtonNotActive, out1 => "DB_MES_Settings_OP70".HMI.MesApproveButton.Color)
   END_RUNG
   RUNG wire#w1
      Contact( "DB_MES_Settings_OP70".HMI.MesApproveButton.Enable )
      Move(in := #cButtonActive, out1 => "DB_MES_Settings_OP70".HMI.MesApproveButton.Color)
   END_RUNG
   RUNG wire#w1
      Contact( FALSE )
      Move(in := #cColorRed, out1 => "DB_MES_Settings_OP70".HMI.MesApproveButton.Color)
   END_RUNG
   RUNG wire#w1
      Contact( "DB_MES_Settings_OP70".HMI.MesApproveButton.Enable )
      Contact( "DB_MES_Settings_OP70".HMI.MesApproveButton.Pressed )
      Move(in := #cColorGreen, out1 => "DB_MES_Settings_OP70".HMI.MesApproveButton.Color)
   END_RUNG
   // the same network as SCL:
   IF TRUE AND NOT "DB_MES_Settings_OP70".HMI.MesApproveButton.Enable THEN
       "DB_MES_Settings_OP70".HMI.MesApproveButton.Color := #cButtonNotActive;
   END_IF;
   IF TRUE AND "DB_MES_Settings_OP70".HMI.MesApproveButton.Enable THEN
       "DB_MES_Settings_OP70".HMI.MesApproveButton.Color := #cButtonActive;
   END_IF;
   IF TRUE AND FALSE THEN "DB_MES_Settings_OP70".HMI.MesApproveButton.Color := #cColorRed; END_IF;
   IF TRUE AND "DB_MES_Settings_OP70".HMI.MesApproveButton.Enable AND "DB_MES_Settings_OP70".HMI.MesApproveButton.Pressed THEN
       "DB_MES_Settings_OP70".HMI.MesApproveButton.Color := #cColorGreen;
   END_IF;
END_REGION

REGION Network 36: MES PopUp: Activation button: Enable
   RUNG wire#powerrail
      Contact( #tEKSLevelOK )
      wire#w1
      Contact( "DB_MES_Settings_OP70".MesDeselected )
      wire#w2
      Coil( "DB_MES_Settings_OP70".HMI.MesActivationButton.Enable )
   END_RUNG
   RUNG wire#w1
      Contact( "DB_MES_Settings_OP70".HMI.MesActivationButton.Pressed )
   END_RUNG wire#w2
   // the same network as SCL:
   "DB_MES_Settings_OP70".HMI.MesActivationButton.Enable := #tEKSLevelOK AND ("DB_MES_Settings_OP70".MesDeselected OR "DB_MES_Settings_OP70".HMI.MesActivationButton.Pressed);
END_REGION

REGION Network 37: MES PopUp: Activation button: Color
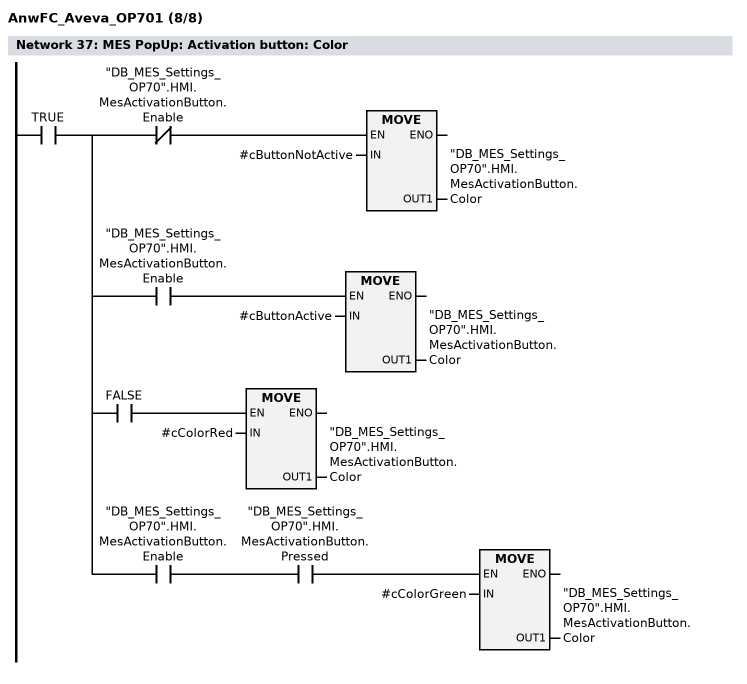
   RUNG wire#powerrail
      Contact( TRUE )
      wire#w1
      I_Contact( "DB_MES_Settings_OP70".HMI.MesActivationButton.Enable )
      Move(in := #cButtonNotActive, out1 => "DB_MES_Settings_OP70".HMI.MesActivationButton.Color)
   END_RUNG
   RUNG wire#w1
      Contact( "DB_MES_Settings_OP70".HMI.MesActivationButton.Enable )
      Move(in := #cButtonActive, out1 => "DB_MES_Settings_OP70".HMI.MesActivationButton.Color)
   END_RUNG
   RUNG wire#w1
      Contact( FALSE )
      Move(in := #cColorRed, out1 => "DB_MES_Settings_OP70".HMI.MesActivationButton.Color)
   END_RUNG
   RUNG wire#w1
      Contact( "DB_MES_Settings_OP70".HMI.MesActivationButton.Enable )
      Contact( "DB_MES_Settings_OP70".HMI.MesActivationButton.Pressed )
      Move(in := #cColorGreen, out1 => "DB_MES_Settings_OP70".HMI.MesActivationButton.Color)
   END_RUNG
   // the same network as SCL:
   IF TRUE AND NOT "DB_MES_Settings_OP70".HMI.MesActivationButton.Enable THEN
       "DB_MES_Settings_OP70".HMI.MesActivationButton.Color := #cButtonNotActive;
   END_IF;
   IF TRUE AND "DB_MES_Settings_OP70".HMI.MesActivationButton.Enable THEN
       "DB_MES_Settings_OP70".HMI.MesActivationButton.Color := #cButtonActive;
   END_IF;
   IF TRUE AND FALSE THEN "DB_MES_Settings_OP70".HMI.MesActivationButton.Color := #cColorRed; END_IF;
   IF TRUE AND "DB_MES_Settings_OP70".HMI.MesActivationButton.Enable AND "DB_MES_Settings_OP70".HMI.MesActivationButton.Pressed THEN
       "DB_MES_Settings_OP70".HMI.MesActivationButton.Color := #cColorGreen;
   END_IF;
END_REGION
END_FUNCTION
